// TIA Portal V17 export
// export: Created 2023-04-11T11:35:16.3671027Z, ExportSetting WithDefaults, DisplayName Totally Integrated Automation Portal, DisplayVersion V17 Update 3, DisplayName TIA Portal Openness, DisplayVersion V17 Update 3, DisplayName TIA Portal Version Control Interface, DisplayVersion V17, DisplayName SINAMICS Startdrive Advanced, DisplayVersion V17 Update2, DisplayName SINAMICS Startdrive G130, G150, S120, S150, SINAMICS MV, S210, DisplayVersion V17 Update2, DisplayName SINAMICS Startdrive G110M, G120, G120C, G120D, G120P, G115D, DisplayVersion V17 Update2, DisplayName STEP 7 Professional, DisplayVersion V17 Update 3, DisplayName STEP 7 Safety, DisplayVersion V17, DisplayName WinCC UA Professional, DisplayVersion V17 Update 3
TYPE "t_IpPort2"
// stored: IsFailsafeCompliant false
   STRUCT
      Ip : Array[0..3] of USInt;
      Port : UInt;
   END_STRUCT;
END_TYPE
